{attribute 'GeneratedUsingTerminal: EL5002-0000-0020'}
{attribute addProperty BoxType "EL5002-0000-0020"}
{attribute addProperty Id "StatusAT %I*Status_C03E24957Counter_valueAT %I*UDINT4"}
{attribute addProperty CRC "3986776708"}
{attribute addProperty Size "11"}
TYPE SSI_Inputs_Channel_EDA16284 :
STRUCT
	{attribute addProperty Name "Status"}
	Status AT %I* : Status_C03E2495;
	{attribute addProperty Name "Counter_value"}
	Counter_value AT %I* : UDINT;
END_STRUCT
END_TYPE

(* stored: Version 1.2.0.0, ProductVersion 3.1.4024.9
   DUT SSI_Inputs_Channel_EDA16284: Id {e08efa9d-5246-458c-9050-c89f3fda3aa3} *)
